FUNCTION_BLOCK FB_CondensingBoilerSystem EXTENDS FB_SystemContinous
VAR_INPUT
END_VAR
VAR_OUTPUT
END_VAR
VAR
	//default parameters
	localDefaultParameters : ST_CondensingBoilerDefaultParameters;

	//condensing boiler
	CondensingBoiler : FB_CondensingBoiler;
	
	// timer for condensing boiler
	bStartTimer_CondensingBoiler : BOOL;
	Timer_CondensingBoiler : TON;
	
	//valves
	ST_SV331DefaultParameters : ST_DiscreteValveDefaultParameters := (nFeedback := 3);
	ST_RV331DefaultParameters :  ST_MixingValveDefaultParameters := (bFeedbackSignal := TRUE, fControllerAmplification := 1, tControllerIntegralTime := T#100S, fOutMinLimit := 50,  tTaskCycleTime := GlobalVariables.tTaskCycleTime_MAIN, tCtrlCycleTime := GlobalVariables.tCtrlCycleTime_MAIN, fOffsetTerminal := 7970);			
	SV331 : FB_DiscreteValve := (ST_DefaultParameters := ST_SV331DefaultParameters);
	RV331 : FB_MixingValve := (ST_DefaultParameters := ST_RV331DefaultParameters);	
	
	//heat counters
	WMZ331 : FB_MollineC3HeatCounter;
	GM331 : FB_GasMeter_Aerius_G4(); //must be implemeted correctly, maybe use FB_MBUS_HYD_PortPulse ?
	
	//internal variables
	bSetStatusOn_CondensingBoiler : BOOL;
	bSetStatusOn_SV331 : BOOL;
	bStatusOn_SV331 : BOOL;
	bSetStatusOn_RV331 : BOOL;
	bStatusOn_RV331 : BOOL;
END_VAR

MAIN();

Timer_CondensingBoiler(IN := bStartTimer_CondensingBoiler,
	PT := T#120S);

CondensingBoiler.GetState();
CondensingBoiler(bSetStatusOnAutomatic := bSetStatusOn_CondensingBoiler,
	bAlgorithmPermission := bAlgorithmPermission,
	fSetPointAutomatic := fSetPoint);
CondensingBoiler.SetState();

SV331.GetState_BI();
SV331(bSetStatusOnAutomatic := bSetStatusOn_SV331,
	bAlgorithmPermission := bAlgorithmPermission);
SV331.SetState_BO();

RV331.GetState_AI();
RV331(bSetStatusOnAutomatic := bSetStatusOn_RV331,
	fSetPointAutomatic := 100,
	bAlgorithmPermission := bAlgorithmPermission,
	nControlModeAutomatic := 0,
	fThermalPowerExternal := WMZ331.fHeatFlowRate);
RV331.SetState_AO();

WMZ331(aHeatCounterTelegramm := Telegramm_WZ_Brennwerttherme);
GM331();

METHOD PROTECTED  CheckError : BOOL
VAR_INPUT
END_VAR
VAR_OUTPUT
	bError : BOOL;
END_VAR
//empty method because condensing boiler has no feedback signal
END_METHOD

METHOD PROTECTED  Operational : BOOL
VAR_INPUT
END_VAR
VAR_OUTPUT
	bSwitchToWorking : BOOL := FALSE;
END_VAR
bSetStatusOn_CondensingBoiler := TRUE;
bSwitchToWorking := TRUE;
END_METHOD

METHOD PROTECTED  RampDown : BOOL
VAR_INPUT
END_VAR
VAR_OUTPUT
	bRampDownFinished : BOOL := FALSE;
END_VAR
bSetStatusOn_CondensingBoiler := FALSE;
bStartTimer_CondensingBoiler := TRUE;

IF Timer_CondensingBoiler.Q THEN
	bSetStatusOn_SV331 := FALSE;
	bSetStatusOn_RV331 := FALSE;
	bStartTimer_CondensingBoiler := FALSE;
	bRampDownFinished := TRUE;
END_IF
END_METHOD

METHOD PROTECTED  RampUp : BOOL
VAR_INPUT
END_VAR
VAR_OUTPUT
	bRampUpFinished : BOOL := FALSE;
END_VAR
bSetStatusOn_SV331 := TRUE;
bSetStatusOn_RV331 := TRUE;
bStartTimer_CondensingBoiler := TRUE;

IF Timer_CondensingBoiler.Q THEN
	bStartTimer_CondensingBoiler := TRUE;
	bStartTimer_CondensingBoiler := FALSE;
	bRampUpFinished := TRUE;
END_IF
END_METHOD

METHOD PROTECTED   SetSetPointLimits : BOOL
VAR_INPUT
END_VAR
aSetPointLimits[1] := localDefaultParameters.aSetPointLimitsTemperature[1];
aSetPointLimits[2] := localDefaultParameters.aSetPointLimitsTemperature[2];
END_METHOD

METHOD PROTECTED  SetState : BOOL
VAR_INPUT
END_VAR
VAR_OUTPUT
END_VAR
fOperatingPoint := WMZ331.fFeedTemperature;

controlState.bStatusOn := bSetStatusOn;
setPointState.aSetPointLimits := aSetPointLimits;
setPointState.fSetPoint := fSetPoint;
setPointState.fOperatingPoint := fOperatingPoint;
setPointState.sSetPointUnit := 'degreeC';
setPointState.sOperatingPointUnit := 'degreeC';
END_METHOD

METHOD PROTECTED  Working : BOOL
VAR_INPUT
END_VAR
VAR_OUTPUT
	bSwitchToOperational : BOOL := FALSE;
END_VAR
//empty method
END_METHOD

END_FUNCTION_BLOCK

(* stored: Version 1.1.0.1, ProductVersion 3.1.4024.10
   POU FB_CondensingBoilerSystem: Id {4ea81eb2-294a-4a5e-96a7-bc4244c6fcae}, SpecialFunc None
   Method CheckError: Id {aa46f833-0868-4c08-bf1e-1e375947cd52}
   Method Operational: Id {89c73f92-8b51-41f6-8362-a0e75414aef8}
   Method RampDown: Id {f4498be3-ce38-4ec5-8af6-38d778115c09}
   Method RampUp: Id {07b676af-72cc-493f-bd50-f12fd9247171}
   Method SetSetPointLimits: Id {f965b277-8513-4b0c-b7ab-3300e3195be6}
   Method SetState: Id {89d56525-651c-4f36-9363-7c8b8df2e26d}
   Method Working: Id {e08c068f-6841-4dc4-9eef-48381b4cb913} *)
